(* IEC 61131-3 sources: moqui-plc/iec61131/moqui/framework/src/main/org/moqui/diagnostics, 14 files *)

(* ---- ResetPolicy.dut ---- *)
(*#-#-#-#-#-#-#-#-#-#---Declaration---#-#-#-#-#-#-#-#-#-#-#-#-#*)

{attribute 'qualified_only'}
{attribute 'strict'}
(* Reset policy bitfields *)
TYPE ResetPolicy : (
	AuxReset := 512,
	UnconditionedReset := 16384,
	AutoConditionedReset := 8192,
	AutoProvisionalReset := 4096,
	AutoPriorityReset := 2048,
	AutoReset := 1024
); END_TYPE

(* ---- ResetPolicy.st ---- *)
(* Reset policy bitfields *)
TYPE ResetPolicy : (
	AuxReset := 512,
	UnconditionedReset := 16384,
	AutoConditionedReset := 8192,
	AutoProvisionalReset := 4096,
	AutoPriorityReset := 2048,
	AutoReset := 1024
); END_TYPE

(* ---- SignalCategory.dut ---- *)
(*#-#-#-#-#-#-#-#-#-#---Declaration---#-#-#-#-#-#-#-#-#-#-#-#-#*)

{attribute 'qualified_only'}
{attribute 'strict'}
(*
 * Signal category bitfields for assigning static priorities (time independent).
 * Maximum priority to alarms, minimum priority to information.
 * A dynamic priority (maximum priority to the first, priority decreasing with time)
 * could be assigned to each signal of the same category, and an additional static priority
 * could be assigned using the signal code in case of simultaneous activation inside the same category.
 * For alarms, anomalies and warnings, both the priority types are available,
 * for information only the second one.
 *)
TYPE SignalCategory : (
    Alarm := 0, (* Critical: Needs manual reset. Examples: emergencies, protections, critical faults, etc. *)
    Anomaly, (* Soft fault: Can be auto-reseted. Examples: light faults, performance degradation, etc. *)
    Warning, (* Notification: Material depletion, supply channels obstruction, etc. *)
    Information (* State info: Operative modes and instructions, machine states, etc. *)
); END_TYPE

(* ---- SignalCategory.st ---- *)
(*
 * Signal category bitfields for assigning static priorities (time independent).
 * Maximum priority to alarms, minimum priority to information.
 * A dynamic priority (maximum priority to the first, priority decreasing with time)
 * could be assigned to each signal of the same category, and an additional static priority
 * could be assigned using the signal code in case of simultaneous activation inside the same category.
 * For alarms, anomalies and warnings, both the priority types are available,
 * for information only the second one.
 *)
TYPE SignalCategory : (
    Alarm := 0, (* Critical: Needs manual reset. Examples: emergencies, protections, critical faults, etc. *)
    Anomaly, (* Soft fault: Can be auto-reseted. Examples: light faults, performance degradation, etc. *)
    Warning, (* Notification: Material depletion, supply channels obstruction, etc. *)
    Information (* State info: Operative modes and instructions, machine states, etc. *)
); END_TYPE

(* ---- SignalMgmtOperatingMode.dut ---- *)
(*#-#-#-#-#-#-#-#-#-#---Declaration---#-#-#-#-#-#-#-#-#-#-#-#-#*)

{attribute 'qualified_only'}
{attribute 'strict'}
TYPE SignalMgmtOperatingMode : (
    Reset := 0, (* Complete reset *)
    Prepare, (* Pre-processing phase where the reset edges valid for the entire scan are prepared *)
    Process (* Evaluate and process the state of a single specific signal *)
); END_TYPE

(* ---- SignalMgmtOperatingMode.st ---- *)
TYPE SignalMgmtOperatingMode : (
    Reset := 0, (* Complete reset *)
    Prepare, (* Pre-processing phase where the reset edges valid for the entire scan are prepared *)
    Process (* Evaluate and process the state of a single specific signal *)
); END_TYPE

(* ---- SignalOutputAction.dut ---- *)
(*#-#-#-#-#-#-#-#-#-#---Declaration---#-#-#-#-#-#-#-#-#-#-#-#-#*)

{attribute 'qualified_only'}
{attribute 'strict'}
(* Signal actions.
 * The definition of each action role is a designer choice.
 *)
TYPE SignalOutputAction : (
	None := 16#0000,
	EmergencyStop := 16#0001,
	ImmediateStop := 16#0002,
	OnPhaseStop := 16#0003,
    Inhibition := 16#0004
	(* etc. *)
) DWORD; END_TYPE

(* ---- SignalOutputAction.st ---- *)
(* Signal actions.
 * The definition of each action role is a designer choice.
 *)
TYPE SignalOutputAction : (
	None := 16#0000,
	EmergencyStop := 16#0001,
	ImmediateStop := 16#0002,
	OnPhaseStop := 16#0003,
    Inhibition := 16#0004
	(* etc. *)
) DWORD; END_TYPE

(* ---- NetworkDiagnostics.pou ---- *)
(*#-#-#-#-#-#-#-#-#-#---Declaration---#-#-#-#-#-#-#-#-#-#-#-#-#*)

{attribute 'no_assign'}
(* Run network diagnostics on the Ethernet adapter and IO modules *)
FUNCTION_BLOCK NetworkDiagnostics
VAR_EXTERNAL
	fieldbus : FieldbusProtocol;
END_VAR
VAR_OUTPUT
	error: BOOL;
END_VAR
VAR
	(* Logger facade *)
	logger : LoggerFacade;
	module : DED.IDevice;
	moduleInfo : DED.DEVICE_INFO;
	moduleName : STRING;
	moduleStatus : DED.DEVICE_STATE;
	moduleError : DED.ERROR;
	diagnosisInfoAvailable : BOOL;
    diagnosisInfoBuffer : STRING;
	fieldbusDataPtr : DED.CAA.PVOID;
	fieldbusdata : POINTER TO STRING;
	dataSize : DED.CAA.SIZE;
    dataCount : DED.CAA.SIZE;
	diagnoseIoModule : RemoteIoModuleDiagnostics;
	i: INT;
	init : BOOL;
END_VAR

(*#-#-#-#-#-#-#-#-#-#---Implementation---#-#-#-#-#-#-#-#-#-#-#-#-#*)

error := TRUE;

IF NOT init THEN
	(* Logger facade init *)
	logger.enable := TRUE; logger.loggerName := 'RunNetworkDiagnostics';
	init := TRUE;
END_IF;

(*
 * CODESYS includes an OPC UA Server that exposes the PLC variables for external clients.
 * Typically, you do not detect the server’s "failure" directly in user logic,
 * because the server is part of the CODESYS runtime.
 *)

(*
 * To enable/disable the ethernet adapter or other devices, use the following reconfigure command:
 *     Ethernet.Enable := TRUE/FALSE;
 *     reconfigure(xExecute := TRUE, itfNode := Ethernet);
*)

logger(message := concat(concat(concat('Run diagnostics on Ethernet adapeter with name: ', ethernet.DeviceName), ' and NIC name: '), ethernet.NICName),
	level := LogLevel.DEBUG);
(* For applications without remote IO modules or with IO modules integrated into the PLC rack. *)
IF NOT ethernet.Enable THEN
	logger(message := 'The Ethernet adapter is disabled.', level := LogLevel.DEBUG);
	NetworkDiagnostics.error := FALSE;
	RETURN;
END_IF;
IF ethernet.ChildNodeCount = 0 THEN
	logger(message := 'No child devices under the Ethernet adapter. Disable the Ethernet adapter!');
END_IF;
IF ethernet.State = IODrvEthernet.EthernetState.ERROR THEN
	logger(message := 'Ethernet adapter in error state.', level := LogLevel.ERROR);
	RETURN;
END_IF;
IF ethernet.State = IODrvEthernet.EthernetState.NOT_CONFIGURED THEN
	logger(message := 'Ethernet adapter not configured.', level := LogLevel.ERROR);
	RETURN;
END_IF;
IF ethernet.State = IODrvEthernet.EthernetState.SET_IP_ERROR THEN
	logger(message := 'Invalid IP address configured for the Ethernet adapter.', level := LogLevel.ERROR);
	RETURN;
END_IF;
IF ethernet.State = IODrvEthernet.EthernetState.DISCONNECTED THEN
	logger(message := 'Ethernet adapter disconnected.', level := LogLevel.ERROR);
	RETURN;
END_IF;

(*
 * Avoid checking software subsystems of the network stack (e.g. Modbus TCP Client component).
 * Check only the physical remote devices.
 * Find the first physical remote device.
 *)
module := DED.INode_TO_IDevice(ethernet.FirstChildNode.FirstChildNode);
FOR i := 1 TO __UXINT_TO_INT(module.SiblingNodeCount) DO
	module := DED.INode_TO_IDevice(module.NextSiblingNode);
	module.GetDeviceInfo(deiInfo := moduleInfo);
	moduleName := DED.GetDeviceNameString(module);

	IF NOT module.Enable THEN
		logger(message := concat(concat('The ', moduleName), ' IO module is disabled.'), level := LogLevel.DEBUG);
		CONTINUE;
	END_IF;
	IF module.ChildNodeCount = 0 THEN
		logger(message := concat(concat('The ', moduleName), ' IO module has no child devices.'), level := LogLevel.DEBUG);
	END_IF;
	moduleStatus := module.GetDeviceState(xDiagnosisinfoAvailable => diagnosisInfoAvailable, eError => moduleError);
	IF moduleStatus = DED.DEVICE_STATE.ERROR THEN
		logger(message := concat(concat(concat(concat('The ', moduleName), ' IO module is in error state.'), ' Error code: '),
			TO_STRING(moduleError)), level := LogLevel.ERROR);
		logger(message := concat(concat(concat(concat(concat('Module info: Type ', TO_STRING(moduleInfo.eType)), ' - Instance number '),
			TO_STRING(moduleInfo.idInstance)), ' - Unique ID '), TO_STRING(moduleInfo.idSystem)), level := LogLevel.ERROR);

		IF diagnosisInfoAvailable THEN
			moduleError := module.GetDeviceDiagnosisInfo(pData := fieldbusDataPtr, szSize := dataSize, szCount => dataCount);
			fieldbusData := fieldbusDataPtr;
			diagnosisInfoBuffer := fieldbusData^;
			logger(message := 'Diagnosis data:', level := LogLevel.ERROR);
			logger(message := concat('Error code: ', TO_STRING(moduleError)), level := LogLevel.ERROR);
			logger(message := concat('Error stack: ', TO_STRING(fieldbusData)), level := LogLevel.ERROR);
		END_IF;
		CONTINUE;
	END_IF;

	(*
     * Check the remote IO module registers for detecting any errors, if needed.
	 * Otherwise, comment out the following code.
     *)
	diagnoseIoModule(moduleName := moduleName, error => error, diagnosisInfo => diagnosisInfoBuffer);
	IF error THEN
		logger(message := 'The remote IO module is connected but has errors.', level := LogLevel.ERROR);
		logger(message := concat('Error stack: ', diagnosisInfoBuffer), level := LogLevel.ERROR);
		CONTINUE;
	END_IF;
END_FOR;

error := FALSE;

(* ---- NetworkDiagnostics.st ---- *)
(* Run network diagnostics on the Ethernet adapter and IO modules *)
FUNCTION_BLOCK NetworkDiagnostics
	VAR_EXTERNAL
		fieldbus : FieldbusProtocol;
	END_VAR
	VAR_OUTPUT
		error: BOOL;
	END_VAR
	VAR
		(* Logger facade *)
		logger : LoggerFacade;
		module : DED.IDevice;
		moduleInfo : DED.DEVICE_INFO;
		moduleName : STRING;
		moduleStatus : DED.DEVICE_STATE;
		moduleError : DED.ERROR;
		diagnosisInfoAvailable : BOOL;
	    diagnosisInfoBuffer : STRING;
		fieldbusDataPtr : DED.CAA.PVOID;
		fieldbusdata : POINTER TO STRING;
		dataSize : DED.CAA.SIZE;
	    dataCount : DED.CAA.SIZE;
		diagnoseIoModule : RemoteIoModuleDiagnostics;
		i: INT;
		init : BOOL;
	END_VAR

	error := TRUE;

	IF NOT init THEN
		(* Logger facade init *)
		logger.enable := TRUE; logger.loggerName := 'RunNetworkDiagnostics';
		init := TRUE;
	END_IF;

	(*
	 * CODESYS includes an OPC UA Server that exposes the PLC variables for external clients.
	 * Typically, you do not detect the server's "failure" directly in user logic,
	 * because the server is part of the CODESYS runtime.
	 *)

	(*
	 * To enable/disable the ethernet adapter or other devices, use the following reconfigure command:
	 *     Ethernet.Enable := TRUE/FALSE;
	 *     reconfigure(xExecute := TRUE, itfNode := Ethernet);
	*)

	logger(message := concat(concat(concat('Run diagnostics on Ethernet adapeter with name: ', ethernet.DeviceName), ' and NIC name: '), ethernet.NICName),
		level := LogLevel.DEBUG);
	(* For applications without remote IO modules or with IO modules integrated into the PLC rack. *)
	IF NOT ethernet.Enable THEN
		logger(message := 'The Ethernet adapter is disabled.', level := LogLevel.DEBUG);
		error := FALSE;
		RETURN;
	END_IF;
	IF ethernet.ChildNodeCount = 0 THEN
		logger(message := 'No child devices under the Ethernet adapter. Disable the Ethernet adapter!');
	END_IF;
	IF ethernet.State = IODrvEthernet.EthernetState.ERROR THEN
		logger(message := 'Ethernet adapter in error state.', level := LogLevel.ERROR);
		RETURN;
	END_IF;
	IF ethernet.State = IODrvEthernet.EthernetState.NOT_CONFIGURED THEN
		logger(message := 'Ethernet adapter not configured.', level := LogLevel.ERROR);
		RETURN;
	END_IF;
	IF ethernet.State = IODrvEthernet.EthernetState.SET_IP_ERROR THEN
		logger(message := 'Invalid IP address configured for the Ethernet adapter.', level := LogLevel.ERROR);
		RETURN;
	END_IF;
	IF ethernet.State = IODrvEthernet.EthernetState.DISCONNECTED THEN
		logger(message := 'Ethernet adapter disconnected.', level := LogLevel.ERROR);
		RETURN;
	END_IF;

	(*
	 * Avoid checking software subsystems of the network stack (e.g. Modbus TCP Client component).
	 * Check only the physical remote devices.
	 * Find the first physical remote device.
	 *)
	module := DED.INode_TO_IDevice(ethernet.FirstChildNode.FirstChildNode);
	FOR i := 1 TO __UXINT_TO_INT(module.SiblingNodeCount) DO
		module := DED.INode_TO_IDevice(module.NextSiblingNode);
		module.GetDeviceInfo(deiInfo := moduleInfo);
		moduleName := DED.GetDeviceNameString(module);

		IF NOT module.Enable THEN
			logger(message := concat(concat('The ', moduleName), ' IO module is disabled.'), level := LogLevel.DEBUG);
			CONTINUE;
		END_IF;
		IF module.ChildNodeCount = 0 THEN
			logger(message := concat(concat('The ', moduleName), ' IO module has no child devices.'), level := LogLevel.DEBUG);
		END_IF;
		moduleStatus := module.GetDeviceState(xDiagnosisinfoAvailable => diagnosisInfoAvailable, eError => moduleError);
		IF moduleStatus = DED.DEVICE_STATE.ERROR THEN
			logger(message := concat(concat(concat(concat('The ', moduleName), ' IO module is in error state.'), ' Error code: '),
				TO_STRING(moduleError)), level := LogLevel.ERROR);
			logger(message := concat(concat(concat(concat(concat('Module info: Type ', TO_STRING(moduleInfo.eType)), ' - Instance number '),
				TO_STRING(moduleInfo.idInstance)), ' - Unique ID '), TO_STRING(moduleInfo.idSystem)), level := LogLevel.ERROR);

			IF diagnosisInfoAvailable THEN
				moduleError := module.GetDeviceDiagnosisInfo(pData := fieldbusDataPtr, szSize := dataSize, szCount => dataCount);
				fieldbusData := fieldbusDataPtr;
				diagnosisInfoBuffer := fieldbusData^;
				logger(message := 'Diagnosis data:', level := LogLevel.ERROR);
				logger(message := concat('Error code: ', TO_STRING(moduleError)), level := LogLevel.ERROR);
				logger(message := concat('Error stack: ', TO_STRING(fieldbusData)), level := LogLevel.ERROR);
			END_IF;
			CONTINUE;
		END_IF;

		(*
	     * Check the remote IO module registers for detecting any errors, if needed.
		 * Otherwise, comment out the following code.
	     *)
		diagnoseIoModule(moduleName := moduleName, error => error, diagnosisInfo => diagnosisInfoBuffer);
		IF error THEN
			logger(message := 'The remote IO module is connected but has errors.', level := LogLevel.ERROR);
			logger(message := concat('Error stack: ', diagnosisInfoBuffer), level := LogLevel.ERROR);
			CONTINUE;
		END_IF;
	END_FOR;

	error := FALSE;
	END_FUNCTION_BLOCK

(* ---- RemoteIoModuleDiagnostics.pou ---- *)
(*#-#-#-#-#-#-#-#-#-#---Declaration---#-#-#-#-#-#-#-#-#-#-#-#-#*)

{attribute 'no_assign'}
FUNCTION_BLOCK RemoteIoModuleDiagnostics
VAR_EXTERNAL
	fieldbus : FieldbusProtocol;
END_VAR
VAR_INPUT
	moduleName : STRING;
END_VAR
VAR_OUTPUT
	error : BOOL;
	diagnosisInfo : STRING;
END_VAR
VAR
	byteArrayBuffer : ARRAY[0..1] OF BYTE;
	(* ABB parameters *)
	deviceState : BYTE;
	parameterState : BYTE;
END_VAR

(*#-#-#-#-#-#-#-#-#-#---Implementation---#-#-#-#-#-#-#-#-#-#-#-#-#*)

error := TRUE;

(*
(* Example diagnostic code *)
IF moduleName = 'io1' THEN
	toByteArray(inputWord := io1DeviceInformationBlock, byteArray => byteArrayBuffer);
	deviceState := byteArrayBuffer[0];
	parameterState := byteArrayBuffer[1];
(*
ELSIF moduleName = 'io2' THEN
	toByteArray(inputWord := io2DeviceInformationBlock, byteArray => byteArrayBuffer);
    deviceState := byteArrayBuffer[0];
    parameterState := byteArrayBuffer[1];
*)
ELSE
	RETURN;
END_IF;

(* The actual state of the remote IO module *)
diagnosisInfo := concat(concat('IO module ', moduleName), ' diagnosis info: ');
CASE deviceState OF
	0 : diagnosisInfo := concat('STATE_PREOP', diagnosisInfo);
	1 : diagnosisInfo := concat('STATE_OPERATION', diagnosisInfo);
	2 : diagnosisInfo := concat('STATE_ERROR', diagnosisInfo); RETURN;
	3 : diagnosisInfo := concat('STATE_IP_ERROR', diagnosisInfo); RETURN;
	4 : diagnosisInfo := concat('STATE_CYCLIC_OPERATION', diagnosisInfo);
ELSE
	RETURN;
END_CASE;

CASE parameterState OF
	0 : diagnosisInfo := concat('PARA_STATE_NO_PARA', diagnosisInfo);
	1 : diagnosisInfo := concat('PARA_STATE_PARA_ACTIVE', diagnosisInfo);
	2 : diagnosisInfo := concat('PARA_STATE_PARA_DONE', diagnosisInfo);
	3 : diagnosisInfo := concat('PARA_STATE_PARA_DONE', diagnosisInfo);
	4 : diagnosisInfo := concat('PARA_STATE_ERROR', diagnosisInfo); RETURN;
ELSE
	RETURN;
END_CASE;

(* etc. *)
*)

error := FALSE;

(* ---- RemoteIoModuleDiagnostics.st ---- *)
FUNCTION_BLOCK RemoteIoModuleDiagnostics
	VAR_EXTERNAL
		fieldbus : FieldbusProtocol;
	END_VAR
	VAR_INPUT
		moduleName : STRING;
	END_VAR
	VAR_OUTPUT
		error : BOOL;
		diagnosisInfo : STRING;
	END_VAR
	VAR
		byteArrayBuffer : ARRAY[0..1] OF BYTE;
		(* ABB parameters *)
		deviceState : BYTE;
		parameterState : BYTE;
	END_VAR

	error := TRUE;

	(*
	(* Example diagnostic code *)
	IF moduleName = 'io1' THEN
		toByteArray(inputWord := io1DeviceInformationBlock, byteArray => byteArrayBuffer);
		deviceState := byteArrayBuffer[0];
		parameterState := byteArrayBuffer[1];
	(*
	ELSIF moduleName = 'io2' THEN
		toByteArray(inputWord := io2DeviceInformationBlock, byteArray => byteArrayBuffer);
	    deviceState := byteArrayBuffer[0];
	    parameterState := byteArrayBuffer[1];
	*)
	ELSE
		RETURN;
	END_IF;

	(* The actual state of the remote IO module *)
	diagnosisInfo := concat(concat('IO module ', moduleName), ' diagnosis info: ');
	CASE deviceState OF
		0 : diagnosisInfo := concat('STATE_PREOP', diagnosisInfo);
		1 : diagnosisInfo := concat('STATE_OPERATION', diagnosisInfo);
		2 : diagnosisInfo := concat('STATE_ERROR', diagnosisInfo); RETURN;
		3 : diagnosisInfo := concat('STATE_IP_ERROR', diagnosisInfo); RETURN;
		4 : diagnosisInfo := concat('STATE_CYCLIC_OPERATION', diagnosisInfo);
	ELSE
		RETURN;
	END_CASE;

	CASE parameterState OF
		0 : diagnosisInfo := concat('PARA_STATE_NO_PARA', diagnosisInfo);
		1 : diagnosisInfo := concat('PARA_STATE_PARA_ACTIVE', diagnosisInfo);
		2 : diagnosisInfo := concat('PARA_STATE_PARA_DONE', diagnosisInfo);
		3 : diagnosisInfo := concat('PARA_STATE_PARA_DONE', diagnosisInfo);
		4 : diagnosisInfo := concat('PARA_STATE_ERROR', diagnosisInfo); RETURN;
	ELSE
		RETURN;
	END_CASE;

	(* etc. *)
	*)

	error := FALSE;
	END_FUNCTION_BLOCK

(* ---- SignalMgmt.pou ---- *)
(*#-#-#-#-#-#-#-#-#-#---Declaration---#-#-#-#-#-#-#-#-#-#-#-#-#*)

{attribute 'no_assign'}
(* Signal supervisor *)
FUNCTION_BLOCK SignalMgmt
VAR_EXTERNAL CONSTANT
	SIGNAL_LIST_MAX_SIZE : UINT;
END_VAR
VAR_INPUT
	operationType : SignalMgmtOperatingMode;
	(* Signal metadata *)
    code : WORD; (* Unique ID for assigning a static priority to signals of the same category *)
	category : SignalCategory; (* Signal type: Static category/priority level + reset policy *)
	resetPol : ResetPolicy := ResetPolicy.UnconditionedReset;
    outputAction : SignalOutputAction := SignalOutputAction.None; (* Response output/action to the signal detection (e.g. ImmediateStop, EmergencyStop, etc.). *)
	(* Activation condition (condition of failure) or trigger policy for the signal, as a boolean expression *)
    activationCondition : BOOL;
	(*
     * Condition for auto conditioned reset for the signal, as a boolean expression (e.g. MachineNotRunning).
     * The reset condition or policy is considered only if an activation policy has
     * been selected during the configuration phase.
	 *)
	autoResetCondition : BOOL;
    (* Reset commands *)
    reset : BOOL; (* Unconditioned manual/external reset *)
    auxReset : BOOL; (* Auxiliary key or command *)
    (* Selective reset *)
    selectiveResetTrigger : BOOL;
    selectiveResetCode : WORD;
    (* Logger name for recording events associated with signals *)
    loggerName : STRING := '';
END_VAR
VAR_OUTPUT
    cumulativeOutputAction : DWORD := SignalOutputAction.None; (* Cumulative output (stop) for the current cycle *)
    activeCategory : SignalCategory; (* Most severe category active *)
    (* Reset availability indicators (updated each cycle in Prepare+Process, for operator feedback) *)
    resetEnable : BOOL; (* TRUE if at least one active signal has cause gone and requires manual reset *)
    auxResetEnable : BOOL; (* TRUE if at least one active signal has cause gone and accepts aux reset *)
	error : BOOL := FALSE;
END_VAR
VAR
	(* Logger facade *)
    logger : LoggerFacade;
    (* Persistent signal log *)
    signalList : ARRAY[1..SIGNAL_LIST_MAX_SIZE] OF BOOL;
    (* Variables for detecting reset edges *)
    resetOld : BOOL;
    resetActivation : BOOL;
    auxResetOld : BOOL;
    auxResetActivation : BOOL;
    selectiveResetOld : BOOL;
    selectiveResetActivation : BOOL;
    requiresManualReset : BOOL;
	i : UINT;
END_VAR

(*#-#-#-#-#-#-#-#-#-#---Implementation---#-#-#-#-#-#-#-#-#-#-#-#-#*)

(* Args validation *)
IF (loggerName = '') THEN error := TRUE; RETURN; END_IF;

(* Logger facade init *)
logger.enable := TRUE; logger.loggerName := loggerName;

CASE operationType OF
    SignalMgmtOperatingMode.Reset :
		logger(message := 'Signal management reset.', level := LogLevel.DEBUG);
        FOR i := 1 TO SIGNAL_LIST_MAX_SIZE DO signalList[i] := FALSE; END_FOR;
        resetOld := FALSE; auxResetOld := FALSE; selectiveResetOld := FALSE;
        cumulativeOutputAction := SignalOutputAction.None;
        activeCategory := SignalCategory.Information;
        resetEnable := FALSE; auxResetEnable := FALSE;

    SignalMgmtOperatingMode.Prepare :
		logger(message := 'Prepare: Init cumulative output bitmask for the current cycle. ', level := LogLevel.DEBUG);
        (* Detection of reset edges valid for the entire cycle  *)
        resetActivation := reset AND NOT resetOld;
        resetOld := reset;
        auxResetActivation := auxReset AND NOT auxResetOld;
        auxResetOld := auxReset;
        selectiveResetActivation := selectiveResetTrigger AND NOT selectiveResetOld;
        selectiveResetOld := selectiveResetTrigger;
        (* Init for the current cycle *)
        cumulativeOutputAction := SignalOutputAction.None;
        activeCategory := SignalCategory.Information;
        resetEnable := FALSE; auxResetEnable := FALSE;

    SignalMgmtOperatingMode.Process :
		logger(message := concat('Process signal: ', WORD_TO_STRING(code)), level := LogLevel.DEBUG);

        (* Bounds check *)
        IF (code < 1) OR (code > SIGNAL_LIST_MAX_SIZE) THEN
            error := TRUE;
            RETURN;
        END_IF;

        (*
         * Determine if manual reset is required.
         * - Alarm, Anomaly: require manual reset unless resetPol = AutoReset
         * - Warning, Information: always auto-reset
         *)
        CASE category OF
            SignalCategory.Alarm, SignalCategory.Anomaly:
                (* Both require manual reset by default; AutoReset policy overrides this *)
                requiresManualReset := (resetPol <> ResetPolicy.AutoReset);
            SignalCategory.Warning, SignalCategory.Information:
                requiresManualReset := FALSE;
        END_CASE;

        (* Check the activation condition *)
        IF activationCondition AND NOT signalList[code] THEN
			signalList[code] := TRUE;
            (* Trigger the logger *)
            logger(enable := TRUE, loggerName := loggerName, level := LogLevel.Fatal,
				message := concat(concat('Signal code: ', WORD_TO_STRING(code)), ' active.'));
        END_IF;

        (*
         * Reset logic.
         * An active signal is reset if the physical cause has disappeared (NOT activationCondition)
         * AND one of the following re-entry conditions occurs, filtered by resetPol:
         *   - Auto-reset (Warning/Information, or Alarm/Anomaly with AutoReset policy)
         *   - Unconditioned manual reset: always allowed for Alarm
         *   - Aux reset: only if resetPol = AuxReset
         *   - Conditioned reset: only if resetPol = AutoConditionedReset / AutoProvisionalReset / AutoPriorityReset
         *   - Selective reset: always allowed (supervisor override)
         *)
        IF NOT activationCondition AND signalList[code] THEN
            IF NOT requiresManualReset THEN
                (* Auto-reset: Anomaly, Warning, Information, or Alarm with AutoReset policy *)
                signalList[code] := FALSE;
            ELSIF resetActivation THEN
                (* Unconditioned manual reset *)
                signalList[code] := FALSE;
            ELSIF auxResetActivation AND (resetPol = ResetPolicy.AuxReset) THEN
                (* Aux reset: only if explicitly configured *)
                signalList[code] := FALSE;
            ELSIF autoResetCondition AND (
                    resetPol = ResetPolicy.AutoConditionedReset OR
                    resetPol = ResetPolicy.AutoProvisionalReset OR
                    resetPol = ResetPolicy.AutoPriorityReset) THEN
                (* Conditioned reset: only if explicitly configured *)
                signalList[code] := FALSE;
            ELSIF selectiveResetActivation AND (selectiveResetCode = code) THEN
                (* Selective reset from external supervision: always allowed *)
                signalList[code] := FALSE;
            END_IF;

            IF NOT signalList[code] THEN
                logger(message := concat(concat('Signal code: ', WORD_TO_STRING(code)), ' reset.'));
            END_IF;
        END_IF;

        (* Cumulative stop bitmask *)
        IF signalList[code] THEN
            cumulativeOutputAction := cumulativeOutputAction OR outputAction;
			logger(message := concat('Signal cumulative output: ', DWORD_TO_STRING(cumulativeOutputAction)));

            (* Track the most severe category active in this cycle *)
            IF category < activeCategory THEN
                activeCategory := category;
            END_IF;
        END_IF;

        (* Reset availability: signal is active, cause is gone, manual reset is required *)
        IF signalList[code] AND NOT activationCondition AND requiresManualReset THEN
            resetEnable := TRUE;
        END_IF;
        IF signalList[code] AND NOT activationCondition AND (resetPol = ResetPolicy.AuxReset) THEN
            auxResetEnable := TRUE;
        END_IF;
END_CASE;

(* ---- SignalMgmt.st ---- *)
(* Signal supervisor *)
FUNCTION_BLOCK SignalMgmt
	VAR_EXTERNAL CONSTANT
		SIGNAL_LIST_MAX_SIZE : UINT;
	END_VAR
	VAR_INPUT
		operationType : SignalMgmtOperatingMode;
		(* Signal metadata *)
	    code : WORD; (* Unique ID for assigning a static priority to signals of the same category *)
		category : SignalCategory; (* Signal type: Static category/priority level + reset policy *)
		resetPol : ResetPolicy := ResetPolicy.UnconditionedReset;
	    outputAction : SignalOutputAction := SignalOutputAction.None; (* Response output/action to the signal detection (e.g. ImmediateStop, EmergencyStop, etc.). *)
		(* Activation condition (condition of failure) or trigger policy for the signal, as a boolean expression *)
	    activationCondition : BOOL;
		(*
	     * Condition for auto conditioned reset for the signal, as a boolean expression (e.g. MachineNotRunning).
	     * The reset condition or policy is considered only if an activation policy has
	     * been selected during the configuration phase.
		 *)
		autoResetCondition : BOOL;
	    (* Reset commands *)
	    reset : BOOL; (* Unconditioned manual/external reset *)
	    auxReset : BOOL; (* Auxiliary key or command *)
	    (* Selective reset *)
	    selectiveResetTrigger : BOOL;
	    selectiveResetCode : WORD;
	    (* Logger name for recording events associated with signals *)
	    loggerName : STRING := '';
	END_VAR
	VAR_OUTPUT
	    cumulativeOutputAction : DWORD := SignalOutputAction.None; (* Cumulative output (stop) for the current cycle *)
	    activeCategory : SignalCategory; (* Most severe category active *)
	    (* Reset availability indicators (updated each cycle in Prepare+Process, for operator feedback) *)
	    resetEnable : BOOL; (* TRUE if at least one active signal has cause gone and requires manual reset *)
	    auxResetEnable : BOOL; (* TRUE if at least one active signal has cause gone and accepts aux reset *)
		error : BOOL := FALSE;
	END_VAR
	VAR
		(* Logger facade *)
	    logger : LoggerFacade;
	    (* Persistent signal log *)
	    signalList : ARRAY[1..SIGNAL_LIST_MAX_SIZE] OF BOOL;
	    (* Variables for detecting reset edges *)
	    resetOld : BOOL;
	    resetActivation : BOOL;
	    auxResetOld : BOOL;
	    auxResetActivation : BOOL;
	    selectiveResetOld : BOOL;
	    selectiveResetActivation : BOOL;
	    requiresManualReset : BOOL;
		i : UINT;
	END_VAR

	(* Args validation *)
	IF (loggerName = '') THEN error := TRUE; RETURN; END_IF;

	(* Logger facade init *)
	logger.enable := TRUE; logger.loggerName := loggerName;

	CASE operationType OF
	    SignalMgmtOperatingMode.Reset :
			logger(message := 'Signal management reset.', level := LogLevel.DEBUG);
	        FOR i := 1 TO SIGNAL_LIST_MAX_SIZE DO signalList[i] := FALSE; END_FOR;
	        resetOld := FALSE; auxResetOld := FALSE; selectiveResetOld := FALSE;
	        cumulativeOutputAction := SignalOutputAction.None;
	        activeCategory := SignalCategory.Information;
	        resetEnable := FALSE; auxResetEnable := FALSE;

	    SignalMgmtOperatingMode.Prepare :
			logger(message := 'Prepare: Init cumulative output bitmask for the current cycle. ', level := LogLevel.DEBUG);
	        (* Detection of reset edges valid for the entire cycle  *)
	        resetActivation := reset AND NOT resetOld;
	        resetOld := reset;
	        auxResetActivation := auxReset AND NOT auxResetOld;
	        auxResetOld := auxReset;
	        selectiveResetActivation := selectiveResetTrigger AND NOT selectiveResetOld;
	        selectiveResetOld := selectiveResetTrigger;
	        (* Init for the current cycle *)
	        cumulativeOutputAction := SignalOutputAction.None;
	        activeCategory := SignalCategory.Information;
	        resetEnable := FALSE; auxResetEnable := FALSE;

	    SignalMgmtOperatingMode.Process :
			logger(message := concat('Process signal: ', WORD_TO_STRING(code)), level := LogLevel.DEBUG);

	        (* Bounds check *)
	        IF (code < 1) OR (code > SIGNAL_LIST_MAX_SIZE) THEN
	            error := TRUE;
	            RETURN;
	        END_IF;

	        (*
	         * Determine if manual reset is required.
	         * - Alarm, Anomaly: require manual reset unless resetPol = AutoReset
	         * - Warning, Information: always auto-reset
	         *)
	        CASE category OF
	            SignalCategory.Alarm, SignalCategory.Anomaly:
	                (* Both require manual reset by default; AutoReset policy overrides this *)
	                requiresManualReset := (resetPol <> ResetPolicy.AutoReset);
	            SignalCategory.Warning, SignalCategory.Information:
	                requiresManualReset := FALSE;
	        END_CASE;

	        (* Check the activation condition *)
	        IF activationCondition AND NOT signalList[code] THEN
				signalList[code] := TRUE;
	            (* Trigger the logger *)
	            logger(enable := TRUE, loggerName := loggerName, level := LogLevel.Fatal,
					message := concat(concat('Signal code: ', WORD_TO_STRING(code)), ' active.'));
	        END_IF;

	        (*
	         * Reset logic.
	         * An active signal is reset if the physical cause has disappeared (NOT activationCondition)
	         * AND one of the following re-entry conditions occurs, filtered by resetPol:
	         *   - Auto-reset (Warning/Information, or Alarm/Anomaly with AutoReset policy)
	         *   - Unconditioned manual reset: always allowed for Alarm
	         *   - Aux reset: only if resetPol = AuxReset
	         *   - Conditioned reset: only if resetPol = AutoConditionedReset / AutoProvisionalReset / AutoPriorityReset
	         *   - Selective reset: always allowed (supervisor override)
	         *)
	        IF NOT activationCondition AND signalList[code] THEN
	            IF NOT requiresManualReset THEN
	                (* Auto-reset: Anomaly, Warning, Information, or Alarm with AutoReset policy *)
	                signalList[code] := FALSE;
	            ELSIF resetActivation THEN
	                (* Unconditioned manual reset *)
	                signalList[code] := FALSE;
	            ELSIF auxResetActivation AND (resetPol = ResetPolicy.AuxReset) THEN
	                (* Aux reset: only if explicitly configured *)
	                signalList[code] := FALSE;
	            ELSIF autoResetCondition AND (
	                    resetPol = ResetPolicy.AutoConditionedReset OR
	                    resetPol = ResetPolicy.AutoProvisionalReset OR
	                    resetPol = ResetPolicy.AutoPriorityReset) THEN
	                (* Conditioned reset: only if explicitly configured *)
	                signalList[code] := FALSE;
	            ELSIF selectiveResetActivation AND (selectiveResetCode = code) THEN
	                (* Selective reset from external supervision: always allowed *)
	                signalList[code] := FALSE;
	            END_IF;

	            IF NOT signalList[code] THEN
	                logger(message := concat(concat('Signal code: ', WORD_TO_STRING(code)), ' reset.'));
	            END_IF;
	        END_IF;

	        (* Cumulative stop bitmask *)
	        IF signalList[code] THEN
	            cumulativeOutputAction := cumulativeOutputAction OR outputAction;
				logger(message := concat('Signal cumulative output: ', DWORD_TO_STRING(cumulativeOutputAction)));

	            (* Track the most severe category active in this cycle *)
	            IF category < activeCategory THEN
	                activeCategory := category;
	            END_IF;
	        END_IF;

	        (* Reset availability: signal is active, cause is gone, manual reset is required *)
	        IF signalList[code] AND NOT activationCondition AND requiresManualReset THEN
	            resetEnable := TRUE;
	        END_IF;
	        IF signalList[code] AND NOT activationCondition AND (resetPol = ResetPolicy.AuxReset) THEN
	            auxResetEnable := TRUE;
	        END_IF;
	END_CASE;
	END_FUNCTION_BLOCK
